PROGRAM FB_RollerConveyors
VAR
END_VAR

GVL_ProcesoPalet.sRollerConveyor.bRollerAlmacen1 := TRUE;
GVL_ProcesoPalet.sRollerConveyor.bRollerAlmacen2 := TRUE;
GVL_ProcesoPalet.sRollerConveyor.bCurvedRollerAlmacen := TRUE;

END_PROGRAM

(* stored: Version 1.1.0.1, ProductVersion 3.1.4024.12
   POU FB_RollerConveyors: Id {934fb174-5cc9-46f2-8626-67d23653f419}, SpecialFunc None *)
